{attribute 'linkalways'} 
{attribute 'no_explicit_call' := 'This FB is a CLASS and must be accessed using methods or properties'}
{attribute 'enable_dynamic_creation'}
FUNCTION_BLOCK _ETcVnFeatureScoreTypeORB EXTENDS EnumDatatypeBase
VAR
	localData : ETcVnFeatureScoreTypeORB;
	activeData : REFERENCE TO ETcVnFeatureScoreTypeORB;
	enumBaseDatatype : _DINT(localData);
END_VAR

METHOD PRIVATE AddLocalEnumeration
VAR_INPUT
	Enumeration : T_MAXSTRING;
	Value : ETcVnFeatureScoreTypeORB;
END_VAR
AddEnumeration(Enumeration, Value);
END_METHOD

PROPERTY PUBLIC Address : PVOID
GET
Address := ADR(activeData);
END_GET
END_PROPERTY

METHOD PUBLIC ClearReference
VAR_INPUT
END_VAR
activeData REF= localData;
SetBaseDatatypeReference();
END_METHOD

METHOD PUBLIC Clone : I_Datatype
VAR
    pClone : POINTER TO _ETcVnFeatureScoreTypeORB;
END_VAR
pClone := __NEW(_ETcVnFeatureScoreTypeORB(InitialValue := Value));
Clone := pClone^;
END_METHOD

METHOD FB_init : BOOL
VAR_INPUT
	bInitRetains : BOOL; // if TRUE, the retain variables are initialized (warm start / cold start)
	bInCopyCode : BOOL;  // if TRUE, the instance afterwards gets moved into the copy code (online change)
	InitialValue : ETcVnFeatureScoreTypeORB;
END_VAR
localData := InitialValue;
AddBaseDatatype(enumBaseDatatype);
ClearReference();

AddLocalEnumeration('TCVN_FST_ORB_HARRIS', ETcVnFeatureScoreTypeORB.TCVN_FST_ORB_HARRIS);
AddLocalEnumeration('TCVN_FST_ORB_FAST', ETcVnFeatureScoreTypeORB.TCVN_FST_ORB_FAST);
END_METHOD

PROPERTY PUBLIC Identifier : T_MAXSTRING
GET
Identifier := 'ETcVnFeatureScoreTypeORB';
END_GET
END_PROPERTY

METHOD IsEnumeratorValueEqual : BOOL
VAR_INPUT
	Enumerator : I_KeyValueForwardEnumerator;
END_VAR
VAR
	storedValue : ETcVnFeatureScoreTypeORB;
END_VAR
IF NOT Enumerator.TryGet(storedValue) THEN
	RETURN;
END_IF

IsEnumeratorValueEqual := storedValue = activeData;
END_METHOD

METHOD PUBLIC MakeReferenceTo
VAR_INPUT
	ReferenceTarget : REFERENCE TO ETcVnFeatureScoreTypeORB;
END_VAR
activeData REF= ReferenceTarget;
SetBaseDatatypeReference();
END_METHOD

METHOD PROTECTED SetBaseDatatypeReference
VAR_INPUT
END_VAR
enumBaseDatatype.MakeReferenceTo(activeData);
END_METHOD

PROPERTY PUBLIC Size : UDINT
GET
Size := SIZEOF(activeData);
END_GET
END_PROPERTY

METHOD TryMakeReferenceTo : BOOL
VAR_INPUT
	Target : I_Datatype;
END_VAR
VAR
	targetAsEnum : I_EnumDatatype;
	pTargetData : POINTER TO ETcVnFeatureScoreTypeORB;
END_VAR
IF NOT Target.TryResolveAsEnumDatatype(targetAsEnum) THEN
	RETURN;
END_IF

IF targetAsEnum.Identifier <> Identifier THEN
	RETURN;
END_IF

pTargetData := Target.Address;
activeData REF= pTargetData^;
SetBaseDatatypeReference();
TryMakeReferenceTo := TRUE;
END_METHOD

PROPERTY PUBLIC Value : ETcVnFeatureScoreTypeORB
GET
Value := activeData;
END_GET
SET
activeData := Value;
END_SET
END_PROPERTY

END_FUNCTION_BLOCK

(* stored: Version 1.1.0.1, ProductVersion 3.1.4024.12
   POU _ETcVnFeatureScoreTypeORB: Id {8fcbf26a-f46d-443b-b848-7649aed1c5b0}, SpecialFunc None
   Folder Constructor: Id {114b81d0-e3b1-4fff-a4f3-73d542a16603}
   Folder Private: Id {308b2b10-38f4-4c58-8131-79fc70ff8e7f}
   Folder Protected: Id {dc38ca09-e710-4ff9-b15a-50840993203b}
   Method AddLocalEnumeration: Id {05321c10-957f-48f4-8e7a-01b36d6ee714}
   Property Address: Id {4921482e-07c5-448e-a8df-cd1914c89a28}
   Get Get: Id {70e3fbbb-d198-453d-a046-850783a09cdc}
   Method ClearReference: Id {8bb14322-91de-4df9-9b02-6a2975f15561}
   Method Clone: Id {fe936426-8fdb-482f-8732-18919b5573cc}
   Method FB_init: Id {d6142206-99d3-4599-8a05-6eb05f2b8809}
   Property Identifier: Id {c266099d-74da-42b9-98ff-6a2a572cce62}
   Get Get: Id {3a29bfa3-6aa0-4502-b538-a28e9b7ddeae}
   Method IsEnumeratorValueEqual: Id {b138eb52-c539-4439-9da5-dbf4352b4e27}
   Method MakeReferenceTo: Id {3aac22e1-1d37-4d2c-9805-84676593c378}
   Method SetBaseDatatypeReference: Id {03f286a2-9915-4a5d-8a38-06a75fc32d1e}
   Property Size: Id {d17ff613-f7fb-4e57-af9e-b946d3fd610f}
   Get Get: Id {9b8f28c4-f3eb-4c1e-8919-784981da1465}
   Method TryMakeReferenceTo: Id {ab4b2fa7-8c73-4860-8d05-e0150f2ef743}
   Property Value: Id {671d40e7-82a9-4fd1-a032-bbda7c3f2e71}
   Get Get: Id {29383bc8-e975-4e7a-970a-5deb2186ecbc}
   Set Set: Id {bcb968a9-afde-4981-ad2a-a9d7c35847f1} *)
